TYPE Integer : LINT; END_TYPE

(* stored: Version 1.1.0.1
   DUT Integer: Id {28080f69-aca8-4ffd-a98e-2aa3100a1bfa} *)
